// Mitsubishi GX Works2 project: 원버튼플립플롭   PLC: Q02/Q02H

PROGRAM MAIN
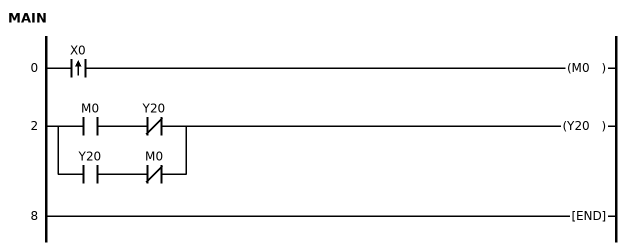
0     LDP     X0
      OUT     M0
2     LD      M0
      ANI     Y20
      LD      Y20
      ANI     M0
      ORB
      OUT     Y20
8     END
END_PROGRAM
